gfCNCPoint6[13263] = {X 14.6334, Y 34.3252, Z -8.0000, A 0.000, B 0.000, C 0.000 }
gfCNCPoint6[13264] = {X 12.2420, Y 34.4773, Z -8.0000, A 0.000, B 0.000, C 0.000 }
gfCNCPoint6[13265] = {X 9.8492, Y 34.6066, Z -8.0000, A 0.000, B 0.000, C 0.000 }
gfCNCPoint6[13266] = {X 8.5942, Y 34.7153, Z -8.0000, A 0.000, B 0.000, C 0.000 }
gfCNCPoint6[13267] = {X 7.3621, Y 34.9773, Z -8.0000, A 0.000, B 0.000, C 0.000 }
gfCNCPoint6[13268] = {X 7.2815, Y 35.1985, Z -8.0000, A 0.000, B 0.000, C 0.000 }
gfCNCPoint6[13269] = {X 7.2536, Y 35.4323, Z -8.0000, A 0.000, B 0.000, C 0.000 }
gfCNCPoint6[13270] = {X 7.3227, Y 35.9818, Z -8.0000, A 0.000, B 0.000, C 0.000 }
gfCNCPoint6[13271] = {X 7.5296, Y 36.4956, Z -8.0000, A 0.000, B 0.000, C 0.000 }
gfCNCPoint6[13272] = {X 7.8604, Y 36.9398, Z -8.0000, A 0.000, B 0.000, C 0.000 }
gfCNCPoint6[13273] = {X 8.2934, Y 37.2851, Z -8.0000, A 0.000, B 0.000, C 0.000 }
gfCNCPoint6[13274] = {X 9.1174, Y 37.7035, Z -8.0000, A 0.000, B 0.000, C 0.000 }
gfCNCPoint6[13275] = {X 9.9944, Y 37.9945, Z -8.0000, A 0.000, B 0.000, C 0.000 }
gfCNCPoint6[13276] = {X 11.3291, Y 38.2411, Z -8.0000, A 0.000, B 0.000, C 0.000 }
gfCNCPoint6[13277] = {X 12.6842, Y 38.3182, Z -8.0000, A 0.000, B 0.000, C 0.000 }
gfCNCPoint6[13278] = {X 14.0382, Y 38.2245, Z -8.0000, A 0.000, B 0.000, C 0.000 }
gfCNCPoint6[13279] = {X 15.3698, Y 37.9615, Z -8.0000, A 0.000, B 0.000, C 0.000 }
gfCNCPoint6[13280] = {X 16.6578, Y 37.5334, Z -8.0000, A 0.000, B 0.000, C 0.000 }
gfCNCPoint6[13281] = {X 18.0872, Y 36.8586, Z -8.0000, A 0.000, B 0.000, C 0.000 }
gfCNCPoint6[13282] = {X 19.4300, Y 36.0248, Z -8.0000, A 0.000, B 0.000, C 0.000 }
gfCNCPoint6[13283] = {X 19.5226, Y 35.1553, Z -8.0000, A 0.000, B 0.000, C 0.000 }
gfCNCPoint6[13284] = {X 19.8019, Y 34.3266, Z -8.0000, A 0.000, B 0.000, C 0.000 }
gfCNCPoint6[13285] = {X 20.2547, Y 33.5784, Z -8.0000, A 0.000, B 0.000, C 0.000 }
gfCNCPoint6[13286] = {X 18.1813, Y 33.9857, Z -8.0000, A 0.000, B 0.000, C 0.000 }
gfCNCPoint6[13287] = {X 16.0816, Y 34.2220, Z -8.0000, A 0.000, B 0.000, C 0.000 }
gfCNCPoint6[13288] = {X 15.3576, Y 34.2746, Z -8.0000, A 0.000, B 0.000, C 0.000 }
gfCNCPoint6[13289] = {X 14.6334, Y 34.3252, Z -8.0000, A 0.000, B 0.000, C 0.000 }
gfCNCPoint6[13290] = {X 14.7699, Y 36.3205, Z -8.0000, A 0.000, B 0.000, C 0.000 }
gfCNCPoint6[13291] = {X 14.7699, Y 36.3205, Z -5.0000, A 0.000, B 0.000, C 0.000 }
gfCNCPoint6[13292] = {X 14.7699, Y 36.3205, Z 11.0000, A 0.000, B 0.000, C 0.000 }
gfCNCPoint6[13293] = {X 15.0797, Y 19.4947, Z 11.0000, A 0.000, B 0.000, C 0.000 }
gfCNCPoint6[13294] = {X 15.0797, Y 19.4947, Z -4.1667, A 0.000, B 0.000, C 0.000 }
gfCNCPoint6[13295] = {X 14.5040, Y 19.3644, Z -4.3248, A 0.000, B 0.000, C 0.000 }
gfCNCPoint6[13296] = {X 13.3045, Y 19.2507, Z -4.6477, A 0.000, B 0.000, C 0.000 }
gfCNCPoint6[13297] = {X 12.0998, Y 19.2681, Z -4.9705, A 0.000, B 0.000, C 0.000 }
gfCNCPoint6[13298] = {X 11.2937, Y 19.3838, Z -5.1887, A 0.000, B 0.000, C 0.000 }
gfCNCPoint6[13299] = {X 10.6069, Y 19.4918, Z -5.3750, A 0.000, B 0.000, C 0.000 }
gfCNCPoint6[13300] = {X 9.8995, Y 19.6145, Z -5.5674, A 0.000, B 0.000, C 0.000 }
gfCNCPoint6[13301] = {X 8.6142, Y 20.0611, Z -5.9320, A 0.000, B 0.000, C 0.000 }
gfCNCPoint6[13302] = {X 7.9831, Y 20.4035, Z -6.1244, A 0.000, B 0.000, C 0.000 }
gfCNCPoint6[13303] = {X 7.9269, Y 20.9151, Z -6.2623, A 0.000, B 0.000, C 0.000 }
gfCNCPoint6[13304] = {X 7.4482, Y 22.1341, Z -6.6132, A 0.000, B 0.000, C 0.000 }
gfCNCPoint6[13305] = {X 7.1412, Y 22.5473, Z -6.7511, A 0.000, B 0.000, C 0.000 }
gfCNCPoint6[13306] = {X 8.7368, Y 22.3421, Z -7.1822, A 0.000, B 0.000, C 0.000 }
gfCNCPoint6[13307] = {X 9.6128, Y 22.2715, Z -7.4176, A 0.000, B 0.000, C 0.000 }
gfCNCPoint6[13308] = {X 11.2206, Y 22.2186, Z -7.8487, A 0.000, B 0.000, C 0.000 }
gfCNCPoint6[13309] = {X 11.5028, Y 22.2087, Z -7.9243, A 0.000, B 0.000, C 0.000 }
gfCNCPoint6[13310] = {X 11.7849, Y 22.1973, Z -8.0000, A 0.000, B 0.000, C 0.000 }
gfCNCPoint6[13311] = {X 14.1113, Y 22.0780, Z -8.0000, A 0.000, B 0.000, C 0.000 }
gfCNCPoint6[13312] = {X 16.4344, Y 21.9080, Z -8.0000, A 0.000, B 0.000, C 0.000 }
gfCNCPoint6[13313] = {X 17.0503, Y 21.8306, Z -8.0000, A 0.000, B 0.000, C 0.000 }
gfCNCPoint6[13314] = {X 17.6515, Y 21.6756, Z -8.0000, A 0.000, B 0.000, C 0.000 }
gfCNCPoint6[13315] = {X 17.6731, Y 21.2169, Z -8.0000, A 0.000, B 0.000, C 0.000 }
gfCNCPoint6[13316] = {X 17.5237, Y 20.7827, Z -8.0000, A 0.000, B 0.000, C 0.000 }
gfCNCPoint6[13317] = {X 17.2244, Y 20.4345, Z -8.0000, A 0.000, B 0.000, C 0.000 }
gfCNCPoint6[13318] = {X 16.3055, Y 19.8939, Z -8.0000, A 0.000, B 0.000, C 0.000 }
gfCNCPoint6[13319] = {X 15.2983, Y 19.5441, Z -8.0000, A 0.000, B 0.000, C 0.000 }
gfCNCPoint6[13320] = {X 13.9732, Y 19.3280, Z -8.0000, A 0.000, B 0.000, C 0.000 }
gfCNCPoint6[13321] = {X 12.6318, Y 19.2743, Z -8.0000, A 0.000, B 0.000, C 0.000 }
gfCNCPoint6[13322] = {X 11.2937, Y 19.3838, Z -8.0000, A 0.000, B 0.000, C 0.000 }
gfCNCPoint6[13323] = {X 10.6069, Y 19.4918, Z -8.0000, A 0.000, B 0.000, C 0.000 }
gfCNCPoint6[13324] = {X 9.2579, Y 19.8407, Z -8.0000, A 0.000, B 0.000, C 0.000 }
gfCNCPoint6[13325] = {X 7.9831, Y 20.4035, Z -8.0000, A 0.000, B 0.000, C 0.000 }
gfCNCPoint6[13326] = {X 7.8308, Y 21.1642, Z -8.0000, A 0.000, B 0.000, C 0.000 }
gfCNCPoint6[13327] = {X 7.5472, Y 21.8862, Z -8.0000, A 0.000, B 0.000, C 0.000 }
gfCNCPoint6[13328] = {X 7.1412, Y 22.5473, Z -8.0000, A 0.000, B 0.000, C 0.000 }
gfCNCPoint6[13329] = {X 9.1770, Y 22.3345, Z -8.0000, A 0.000, B 0.000, C 0.000 }
gfCNCPoint6[13330] = {X 11.2206, Y 22.2186, Z -8.0000, A 0.000, B 0.000, C 0.000 }
gfCNCPoint6[13331] = {X 11.5028, Y 22.2083, Z -8.0000, A 0.000, B 0.000, C 0.000 }
gfCNCPoint6[13332] = {X 11.7849, Y 22.1973, Z -8.0000, A 0.000, B 0.000, C 0.000 }
gfCNCPoint6[13333] = {X 7.7926, Y 22.0896, Z -8.0000, A 0.000, B 0.000, C 0.000 }
gfCNCPoint6[13334] = {X 11.7882, Y 22.2773, Z -8.0000, A 0.000, B 0.000, C 0.000 }
gfCNCPoint6[13335] = {X 14.1136, Y 22.1580, Z -8.0000, A 0.000, B 0.000, C 0.000 }
gfCNCPoint6[13336] = {X 16.4358, Y 21.9881, Z -8.0000, A 0.000, B 0.000, C 0.000 }
gfCNCPoint6[13337] = {X 17.0852, Y 21.9053, Z -8.0000, A 0.000, B 0.000, C 0.000 }
gfCNCPoint6[13338] = {X 17.7180, Y 21.7378, Z -8.0000, A 0.000, B 0.000, C 0.000 }
gfCNCPoint6[13339] = {X 17.7562, Y 21.2347, Z -8.0000, A 0.000, B 0.000, C 0.000 }
gfCNCPoint6[13340] = {X 17.6000, Y 20.7550, Z -8.0000, A 0.000, B 0.000, C 0.000 }
gfCNCPoint6[13341] = {X 17.2729, Y 20.3708, Z -8.0000, A 0.000, B 0.000, C 0.000 }
gfCNCPoint6[13342] = {X 16.3395, Y 19.8215, Z -8.0000, A 0.000, B 0.000, C 0.000 }
gfCNCPoint6[13343] = {X 15.3165, Y 19.4662, Z -8.0000, A 0.000, B 0.000, C 0.000 }
gfCNCPoint6[13344] = {X 13.9815, Y 19.2484, Z -8.0000, A 0.000, B 0.000, C 0.000 }
gfCNCPoint6[13345] = {X 12.6299, Y 19.1943, Z -8.0000, A 0.000, B 0.000, C 0.000 }
gfCNCPoint6[13346] = {X 11.2818, Y 19.3047, Z -8.0000, A 0.000, B 0.000, C 0.000 }
gfCNCPoint6[13347] = {X 10.5939, Y 19.4128, Z -8.0000, A 0.000, B 0.000, C 0.000 }
gfCNCPoint6[13348] = {X 9.2120, Y 19.7720, Z -8.0000, A 0.000, B 0.000, C 0.000 }
gfCNCPoint6[13349] = {X 7.9079, Y 20.3534, Z -8.0000, A 0.000, B 0.000, C 0.000 }
gfCNCPoint6[13350] = {X 7.7435, Y 21.1767, Z -8.0000, A 0.000, B 0.000, C 0.000 }
gfCNCPoint6[13351] = {X 7.4230, Y 21.9526, Z -8.0000, A 0.000, B 0.000, C 0.000 }
gfCNCPoint6[13352] = {X 6.9585, Y 22.6519, Z -8.0000, A 0.000, B 0.000, C 0.000 }
gfCNCPoint6[13353] = {X 9.0865, Y 22.4222, Z -8.0000, A 0.000, B 0.000, C 0.000 }
gfCNCPoint6[13354] = {X 11.2233, Y 22.2986, Z -8.0000, A 0.000, B 0.000, C 0.000 }
gfCNCPoint6[13355] = {X 11.5057, Y 22.2883, Z -8.0000, A 0.000, B 0.000, C 0.000 }
gfCNCPoint6[13356] = {X 11.7882, Y 22.2773, Z -8.0000, A 0.000, B 0.000, C 0.000 }
gfCNCPoint6[13357] = {X 15.7556, Y 21.7682, Z -8.0000, A 0.000, B 0.000, C 0.000 }
gfCNCPoint6[13358] = {X 7.7958, Y 22.1696, Z -8.0000, A 0.000, B 0.000, C 0.000 }
gfCNCPoint6[13359] = {X 11.7914, Y 22.3572, Z -8.0000, A 0.000, B 0.000, C 0.000 }
gfCNCPoint6[13360] = {X 14.1181, Y 22.2379, Z -8.0000, A 0.000, B 0.000, C 0.000 }
gfCNCPoint6[13361] = {X 16.4416, Y 22.0679, Z -8.0000, A 0.000, B 0.000, C 0.000 }
gfCNCPoint6[13362] = {X 17.1214, Y 21.9797, Z -8.0000, A 0.000, B 0.000, C 0.000 }
gfCNCPoint6[13363] = {X 17.7830, Y 21.8002, Z -8.0000, A 0.000, B 0.000, C 0.000 }
gfCNCPoint6[13364] = {X 17.8386, Y 21.2529, Z -8.0000, A 0.000, B 0.000, C 0.000 }
gfCNCPoint6[13365] = {X 17.6762, Y 20.7275, Z -8.0000, A 0.000, B 0.000, C 0.000 }
gfCNCPoint6[13366] = {X 17.3214, Y 20.3071, Z -8.0000, A 0.000, B 0.000, C 0.000 }
gfCNCPoint6[13367] = {X 16.3736, Y 19.7491, Z -8.0000, A 0.000, B 0.000, C 0.000 }
gfCNCPoint6[13368] = {X 15.3346, Y 19.3883, Z -8.0000, A 0.000, B 0.000, C 0.000 }
gfCNCPoint6[13369] = {X 13.9897, Y 19.1688, Z -8.0000, A 0.000, B 0.000, C 0.000 }
gfCNCPoint6[13370] = {X 12.6281, Y 19.1143, Z -8.0000, A 0.000, B 0.000, C 0.000 }
gfCNCPoint6[13371] = {X 11.2699, Y 19.2256, Z -8.0000, A 0.000, B 0.000, C 0.000 }
gfCNCPoint6[13372] = {X 10.5808, Y 19.3339, Z -8.0000, A 0.000, B 0.000, C 0.000 }
gfCNCPoint6[13373] = {X 9.6302, Y 19.5540, Z -8.0000, A 0.000, B 0.000, C 0.000 }
gfCNCPoint6[13374] = {X 8.7101, Y 19.8787, Z -8.0000, A 0.000, B 0.000, C 0.000 }
gfCNCPoint6[13375] = {X 7.8319, Y 20.3040, Z -8.0000, A 0.000, B 0.000, C 0.000 }
gfCNCPoint6[13376] = {X 7.8283, Y 20.3454, Z -8.0000, A 0.000, B 0.000, C 0.000 }
gfCNCPoint6[13377] = {X 7.6463, Y 21.2197, Z -8.0000, A 0.000, B 0.000, C 0.000 }
gfCNCPoint6[13378] = {X 7.2852, Y 22.0364, Z -8.0000, A 0.000, B 0.000, C 0.000 }
gfCNCPoint6[13379] = {X 6.7611, Y 22.7594, Z -8.0000, A 0.000, B 0.000, C 0.000 }
gfCNCPoint6[13380] = {X 8.9886, Y 22.5107, Z -8.0000, A 0.000, B 0.000, C 0.000 }
gfCNCPoint6[13381] = {X 11.2260, Y 22.3785, Z -8.0000, A 0.000, B 0.000, C 0.000 }
gfCNCPoint6[13382] = {X 11.5087, Y 22.3682, Z -8.0000, A 0.000, B 0.000, C 0.000 }
gfCNCPoint6[13383] = {X 11.7914, Y 22.3572, Z -8.0000, A 0.000, B 0.000, C 0.000 }
gfCNCPoint6[13384] = {X 15.7589, Y 21.8482, Z -8.0000, A 0.000, B 0.000, C 0.000 }
gfCNCPoint6[13385] = {X 7.7990, Y 22.2495, Z -8.0000, A 0.000, B 0.000, C 0.000 }
gfCNCPoint6[13386] = {X 11.7946, Y 22.4371, Z -8.0000, A 0.000, B 0.000, C 0.000 }
gfCNCPoint6[13387] = {X 14.1226, Y 22.3178, Z -8.0000, A 0.000, B 0.000, C 0.000 }
gfCNCPoint6[13388] = {X 16.4474, Y 22.1477, Z -8.0000, A 0.000, B 0.000, C 0.000 }
gfCNCPoint6[13389] = {X 17.1571, Y 22.0541, Z -8.0000, A 0.000, B 0.000, C 0.000 }
gfCNCPoint6[13390] = {X 17.8467, Y 21.8626, Z -8.0000, A 0.000, B 0.000, C 0.000 }
gfCNCPoint6[13391] = {X 17.9251, Y 21.4213, Z -8.0000, A 0.000, B 0.000, C 0.000 }
gfCNCPoint6[13392] = {X 17.8659, Y 20.9771, Z -8.0000, A 0.000, B 0.000, C 0.000 }
gfCNCPoint6[13393] = {X 17.6748, Y 20.5717, Z -8.0000, A 0.000, B 0.000, C 0.000 }
gfCNCPoint6[13394] = {X 17.3698, Y 20.2434, Z -8.0000, A 0.000, B 0.000, C 0.000 }
gfCNCPoint6[13395] = {X 16.4076, Y 19.6767, Z -8.0000, A 0.000, B 0.000, C 0.000 }
gfCNCPoint6[13396] = {X 15.3528, Y 19.3104, Z -8.0000, A 0.000, B 0.000, C 0.000 }
gfCNCPoint6[13397] = {X 13.9979, Y 19.0892, Z -8.0000, A 0.000, B 0.000, C 0.000 }
gfCNCPoint6[13398] = {X 12.6262, Y 19.0343, Z -8.0000, A 0.000, B 0.000, C 0.000 }
gfCNCPoint6[13399] = {X 11.2580, Y 19.1465, Z -8.0000, A 0.000, B 0.000, C 0.000 }
gfCNCPoint6[13400] = {X 10.5678, Y 19.2550, Z -8.0000, A 0.000, B 0.000, C 0.000 }
gfCNCPoint6[13401] = {X 9.5946, Y 19.4811, Z -8.0000, A 0.000, B 0.000, C 0.000 }
gfCNCPoint6[13402] = {X 8.6532, Y 19.8158, Z -8.0000, A 0.000, B 0.000, C 0.000 }
gfCNCPoint6[13403] = {X 7.7557, Y 20.2549, Z -8.0000, A 0.000, B 0.000, C 0.000 }
gfCNCPoint6[13404] = {X 7.7492, Y 20.3328, Z -8.0000, A 0.000, B 0.000, C 0.000 }
gfCNCPoint6[13405] = {X 7.5473, Y 21.2642, Z -8.0000, A 0.000, B 0.000, C 0.000 }
gfCNCPoint6[13406] = {X 7.1388, Y 22.1252, Z -8.0000, A 0.000, B 0.000, C 0.000 }
gfCNCPoint6[13407] = {X 6.5450, Y 22.8706, Z -8.0000, A 0.000, B 0.000, C 0.000 }
gfCNCPoint6[13408] = {X 8.8812, Y 22.6003, Z -8.0000, A 0.000, B 0.000, C 0.000 }
gfCNCPoint6[13409] = {X 11.2287, Y 22.4585, Z -8.0000, A 0.000, B 0.000, C 0.000 }
gfCNCPoint6[13410] = {X 11.5117, Y 22.4482, Z -8.0000, A 0.000, B 0.000, C 0.000 }
gfCNCPoint6[13411] = {X 11.7946, Y 22.4371, Z -8.0000, A 0.000, B 0.000, C 0.000 }
gfCNCPoint6[13412] = {X 15.7621, Y 21.9281, Z -8.0000, A 0.000, B 0.000, C 0.000 }
gfCNCPoint6[13413] = {X 7.8022, Y 22.3294, Z -8.0000, A 0.000, B 0.000, C 0.000 }
gfCNCPoint6[13414] = {X 11.7978, Y 22.5171, Z -8.0000, A 0.000, B 0.000, C 0.000 }
gfCNCPoint6[13415] = {X 14.1271, Y 22.3976, Z -8.0000, A 0.000, B 0.000, C 0.000 }
gfCNCPoint6[13416] = {X 16.4532, Y 22.2275, Z -8.0000, A 0.000, B 0.000, C 0.000 }
gfCNCPoint6[13417] = {X 17.1922, Y 22.1286, Z -8.0000, A 0.000, B 0.000, C 0.000 }
gfCNCPoint6[13418] = {X 17.9094, Y 21.9251, Z -8.0000, A 0.000, B 0.000, C 0.000 }
gfCNCPoint6[13419] = {X 18.0042, Y 21.4518, Z -8.0000, A 0.000, B 0.000, C 0.000 }
gfCNCPoint6[13420] = {X 17.9478, Y 20.9725, Z -8.0000, A 0.000, B 0.000, C 0.000 }
gfCNCPoint6[13421] = {X 17.7459, Y 20.5341, Z -8.0000, A 0.000, B 0.000, C 0.000 }
gfCNCPoint6[13422] = {X 17.4182, Y 20.1797, Z -8.0000, A 0.000, B 0.000, C 0.000 }
gfCNCPoint6[13423] = {X 16.4416, Y 19.6043, Z -8.0000, A 0.000, B 0.000, C 0.000 }
gfCNCPoint6[13424] = {X 15.3709, Y 19.2325, Z -8.0000, A 0.000, B 0.000, C 0.000 }
gfCNCPoint6[13425] = {X 14.0061, Y 19.0097, Z -8.0000, A 0.000, B 0.000, C 0.000 }
gfCNCPoint6[13426] = {X 12.6243, Y 18.9543, Z -8.0000, A 0.000, B 0.000, C 0.000 }
gfCNCPoint6[13427] = {X 11.2461, Y 19.0674, Z -8.0000, A 0.000, B 0.000, C 0.000 }
gfCNCPoint6[13428] = {X 10.5547, Y 19.1760, Z -8.0000, A 0.000, B 0.000, C 0.000 }
gfCNCPoint6[13429] = {X 9.5589, Y 19.4082, Z -8.0000, A 0.000, B 0.000, C 0.000 }
gfCNCPoint6[13430] = {X 8.5962, Y 19.7531, Z -8.0000, A 0.000, B 0.000, C 0.000 }
gfCNCPoint6[13431] = {X 7.6795, Y 20.2061, Z -8.0000, A 0.000, B 0.000, C 0.000 }
gfCNCPoint6[13432] = {X 7.6695, Y 20.3256, Z -8.0000, A 0.000, B 0.000, C 0.000 }
gfCNCPoint6[13433] = {X 7.5231, Y 21.0759, Z -8.0000, A 0.000, B 0.000, C 0.000 }
gfCNCPoint6[13434] = {X 7.2394, Y 21.7859, Z -8.0000, A 0.000, B 0.000, C 0.000 }
gfCNCPoint6[13435] = {X 6.8281, Y 22.4303, Z -8.0000, A 0.000, B 0.000, C 0.000 }
gfCNCPoint6[13436] = {X 6.3038, Y 22.9868, Z -8.0000, A 0.000, B 0.000, C 0.000 }
gfCNCPoint6[13437] = {X 8.7612, Y 22.6913, Z -8.0000, A 0.000, B 0.000, C 0.000 }
gfCNCPoint6[13438] = {X 11.2315, Y 22.5384, Z -8.0000, A 0.000, B 0.000, C 0.000 }
gfCNCPoint6[13439] = {X 11.5147, Y 22.5281, Z -8.0000, A 0.000, B 0.000, C 0.000 }
gfCNCPoint6[13440] = {X 11.7978, Y 22.5171, Z -8.0000, A 0.000, B 0.000, C 0.000 }
gfCNCPoint6[13441] = {X 15.7653, Y 22.0080, Z -8.0000, A 0.000, B 0.000, C 0.000 }
gfCNCPoint6[13442] = {X 11.7260, Y 22.6000, Z -8.0000, A 0.000, B 0.000, C 0.000 }
gfCNCPoint6[13443] = {X 11.8011, Y 22.5970, Z -8.0000, A 0.000, B 0.000, C 0.000 }
gfCNCPoint6[13444] = {X 14.1316, Y 22.4775, Z -8.0000, A 0.000, B 0.000, C 0.000 }
gfCNCPoint6[13445] = {X 16.4590, Y 22.3073, Z -8.0000, A 0.000, B 0.000, C 0.000 }
gfCNCPoint6[13446] = {X 17.2268, Y 22.2031, Z -8.0000, A 0.000, B 0.000, C 0.000 }
gfCNCPoint6[13447] = {X 17.9710, Y 21.9877, Z -8.0000, A 0.000, B 0.000, C 0.000 }
gfCNCPoint6[13448] = {X 18.0828, Y 21.4826, Z -8.0000, A 0.000, B 0.000, C 0.000 }
gfCNCPoint6[13449] = {X 18.0296, Y 20.9681, Z -8.0000, A 0.000, B 0.000, C 0.000 }
gfCNCPoint6[13450] = {X 17.8170, Y 20.4965, Z -8.0000, A 0.000, B 0.000, C 0.000 }
gfCNCPoint6[13451] = {X 17.4665, Y 20.1160, Z -8.0000, A 0.000, B 0.000, C 0.000 }
gfCNCPoint6[13452] = {X 16.4756, Y 19.5319, Z -8.0000, A 0.000, B 0.000, C 0.000 }
gfCNCPoint6[13453] = {X 15.3891, Y 19.1546, Z -8.0000, A 0.000, B 0.000, C 0.000 }
gfCNCPoint6[13454] = {X 14.0143, Y 18.9301, Z -8.0000, A 0.000, B 0.000, C 0.000 }
gfCNCPoint6[13455] = {X 12.6225, Y 18.8744, Z -8.0000, A 0.000, B 0.000, C 0.000 }
gfCNCPoint6[13456] = {X 11.2342, Y 18.9883, Z -8.0000, A 0.000, B 0.000, C 0.000 }
gfCNCPoint6[13457] = {X 10.5417, Y 19.0971, Z -8.0000, A 0.000, B 0.000, C 0.000 }
gfCNCPoint6[13458] = {X 9.5231, Y 19.3353, Z -8.0000, A 0.000, B 0.000, C 0.000 }
gfCNCPoint6[13459] = {X 8.5392, Y 19.6904, Z -8.0000, A 0.000, B 0.000, C 0.000 }
gfCNCPoint6[13460] = {X 7.6032, Y 20.1575, Z -8.0000, A 0.000, B 0.000, C 0.000 }
gfCNCPoint6[13461] = {X 7.5898, Y 20.3183, Z -8.0000, A 0.000, B 0.000, C 0.000 }
gfCNCPoint6[13462] = {X 7.4463, Y 21.0538, Z -8.0000, A 0.000, B 0.000, C 0.000 }
gfCNCPoint6[13463] = {X 7.1680, Y 21.7496, Z -8.0000, A 0.000, B 0.000, C 0.000 }
gfCNCPoint6[13464] = {X 6.7649, Y 22.3813, Z -8.0000, A 0.000, B 0.000, C 0.000 }
gfCNCPoint6[13465] = {X 6.2510, Y 22.9267, Z -8.0000, A 0.000, B 0.000, C 0.000 }
gfCNCPoint6[13466] = {X 6.2086, Y 22.9635, Z -8.0000, A 0.000, B 0.000, C 0.000 }
gfCNCPoint6[13467] = {X 6.1658, Y 22.9996, Z -8.0000, A 0.000, B 0.000, C 0.000 }
gfCNCPoint6[13468] = {X 6.1511, Y 23.0909, Z -8.0000, A 0.000, B 0.000, C 0.000 }
gfCNCPoint6[13469] = {X 6.2334, Y 23.0783, Z -8.0000, A 0.000, B 0.000, C 0.000 }
gfCNCPoint6[13470] = {X 6.3157, Y 23.0659, Z -8.0000, A 0.000, B 0.000, C 0.000 }
gfCNCPoint6[13471] = {X 8.7685, Y 22.7710, Z -8.0000, A 0.000, B 0.000, C 0.000 }
gfCNCPoint6[13472] = {X 11.2342, Y 22.6184, Z -8.0000, A 0.000, B 0.000, C 0.000 }
gfCNCPoint6[13473] = {X 11.5176, Y 22.6081, Z -8.0000, A 0.000, B 0.000, C 0.000 }
gfCNCPoint6[13474] = {X 11.8011, Y 22.5970, Z -8.0000, A 0.000, B 0.000, C 0.000 }
gfCNCPoint6[13475] = {X 11.7204, Y 20.5986, Z -8.0000, A 0.000, B 0.000, C 0.000 }
gfCNCPoint6[13476] = {X 11.7204, Y 20.5986, Z -5.0000, A 0.000, B 0.000, C 0.000 }
gfCNCPoint6[13477] = {X 11.7204, Y 20.5986, Z 11.0000, A 0.000, B 0.000, C 0.000 }

ENDDAT
